(* IEC 61131-3 sources: Industry-PLC-LLM/data/PLCBEAD_repo/PLCBEAD_PLCEmbed-main/PLC-BEAD/Source/GEB/building_SWITCH_X, 1 file *)

(* ---- SWITCH_X.ST ---- *)
FUNCTION_BLOCK SWITCH_X_Block

	VAR_INPUT
		IN1 :	BOOL;
		IN2 :	BOOL;
		IN3 :	BOOL;
		IN4 :	BOOL;
		IN5 :	BOOL;
		IN6 :	BOOL;
		T_DEBOUNCE :	TIME := T#50ms;
	END_VAR

	VAR_OUTPUT
		Q1 :	BOOL;
		Q2 :	BOOL;
		Q3 :	BOOL;
		Q4 :	BOOL;
		Q5 :	BOOL;
		Q6 :	BOOL;
		Q31 :	BOOL;
		Q41 :	BOOL;
		Q51 :	BOOL;
		Q61 :	BOOL;
		Q32 :	BOOL;
		Q42 :	BOOL;
		Q52 :	BOOL;
		Q62 :	BOOL;
	END_VAR

	VAR
		INIT :	BOOL;
		T1 :	TOF;
		T2 :	TOF;
		T3 :	TOF;
		T4 :	TOF;
		T5 :	TOF;
		T6 :	TOF;
		TX :	TIME;
		X1 :	BOOL;
		X2 :	BOOL;
		E1 :	BOOL;
		E2 :	BOOL;
	END_VAR

	IF NOT init THEN
		init := TRUE;
		IF t_debounce < t#50ms THEN TX := t#50ms; ELSE TX := t_debounce; END_IF;
		T1(PT := TX);
		T2(PT := TX);
		T3(PT := TX);
		T4(PT := TX);
		T5(PT := TX);
		T6(PT := TX);
	ELSE
		Q1 := FALSE;
		Q2 := FALSE;
		Q3 := FALSE;
		Q4 := FALSE;
		Q5 := FALSE;
		Q6 := FALSE;
		Q31 := FALSE;
		Q41 := FALSE;
		Q51 := FALSE;
		Q61 := FALSE;
		Q32 := FALSE;
		Q42 := FALSE;
		Q52 := FALSE;
		Q62 := FALSE;
	END_IF;

		T1(IN := IN1);
		T2(IN := IN2);
		T3(IN := IN3);
		T4(IN := IN4);
		T5(IN := IN5);
		T6(IN := IN6);

	IF t1.Q AND NOT E1 THEN X1 := TRUE; END_IF;
	IF t2.Q AND NOT E2 THEN X2 := TRUE; END_IF;

	IF t1.Q THEN
		IF t3.q THEN
			q31 := TRUE;
			X1 := FALSE;
		ELSIF t4.q THEN
			q41 := TRUE;
			X1 := FALSE;
		ELSIF t5.q THEN
			q51 := TRUE;
			X1 := FALSE;
		ELSIF t6.q THEN
			q61 := TRUE;
			X1 := FALSE;
		END_IF;
	ELSIF t2.Q THEN
		IF t3.q THEN
			q32 := TRUE;
			X2 := FALSE;
		ELSIF t4.q THEN
			q42 := TRUE;
			X2 := FALSE;
		ELSIF t5.q THEN
			q52 := TRUE;
			X2 := FALSE;
		ELSIF t6.q THEN
			q62 := TRUE;
			X2 := FALSE;
		END_IF;
	ELSIF NOT T1.Q AND E1 AND X1 THEN
		Q1 := TRUE;
		X1 := FALSE;
	ELSIF NOT T2.Q AND E2 AND X2 THEN
		Q2 := TRUE;
		X2 := FALSE;
	ELSIF T3.Q THEN
		Q3 := TRUE;
	ELSIF T4.Q THEN
		Q4 := TRUE;
	ELSIF T5.Q THEN
		Q5 := TRUE;
	ELSIF T6.Q THEN
		Q6 := TRUE;
	END_IF;

	E1 := T1.Q;
	E2 := T2.Q;
END_FUNCTION_BLOCK

PROGRAM program0
	VAR
		IN1 :	BOOL;
		IN2 :	BOOL;
		IN3 :	BOOL;
		IN4 :	BOOL;
		IN5 :	BOOL;
		IN6 :	BOOL;
		T_DEBOUNCE :	TIME := T#50ms;
		Q1 :	BOOL;
		Q2 :	BOOL;
		Q3 :	BOOL;
		Q4 :	BOOL;
		Q5 :	BOOL;
		Q6 :	BOOL;
		Q31 :	BOOL;
		Q41 :	BOOL;
		Q51 :	BOOL;
		Q61 :	BOOL;
		Q32 :	BOOL;
		Q42 :	BOOL;
		Q52 :	BOOL;
		Q62 :	BOOL;

		func_block : SWITCH_X_Block;
	END_VAR
	func_block.IN1 := IN1;
	func_block.IN2 := IN2;
	func_block.IN3 := IN3 ;
	func_block.IN4 := IN4;
	func_block.IN5 := IN5;
	func_block.IN6 := IN6 ;
	func_block.T_DEBOUNCE := T_DEBOUNCE;

	func_block();
	Q1  := func_block.Q1;
	Q2  := func_block.Q2;
	Q3  := func_block.Q3;
	Q4  := func_block.Q4;
	Q5  := func_block.Q5;
	Q6  := func_block.Q6;
	Q31  := func_block.Q31;
	Q41  := func_block.Q41;
	Q51  := func_block.Q51;
	Q61  := func_block.Q61;
	Q32  := func_block.Q32;
	Q42  := func_block.Q42;
	Q52  := func_block.Q52;
	Q62  := func_block.Q62;

END_PROGRAM
